# EPICS IOC start-up script: ipApp/iocsh/LakeShore_218.iocsh
# ### LakeShore_330.iocsh ###

#- ###################################################
#- PREFIX         - IOC Prefix
#- INSTANCE       - Instance Prefix
#- PORT           - Serial port name
#- IP             - Location of IP module
#- ###################################################

iocshLoad("$(IP)/iocsh/setSerialParams.iocsh", "PORT=$(PORT), BAUD=9600, BITS=7, STOP=1, PARITY=none")

asynOctetSetInputEos( "$(PORT)", -1, "\n")
asynOctetSetOutputEos("$(PORT)", -1, "\n")

dbLoadRecords("$(IP)/ipApp/Db/LakeShore218.vdb", "P=$(PREFIX),R=$(INSTANCE),PORT=$(PORT)")
